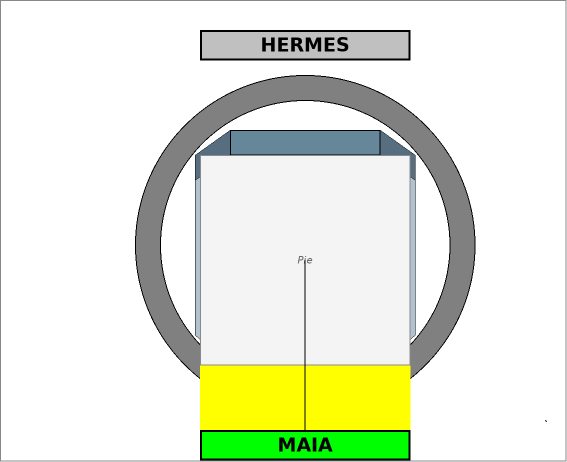
VISUALIZATION VISU_M3RotationFigure_1  // 567x462
    Ellipse (135,75 340x340)
    Ellipse (160,100 290x290)
    Polygon (545,420) (546,421)
    Polygon (230,155) (195,180) (195,155) (230,130) (380,130) (415,155) (415,180) (380,155)
    Polygon (230,365) (195,335) (195,180) (230,155) (380,155) (415,180) (415,335) (380,365)
    Line (565,390)
    Rectangle (230,130 150x25)
    Rectangle (200,260 210x200)
    Pie (200,155 210x210)
    Line (305,445) (305,260)
    Rectangle (200,430 210x30), "MAIA"
    Rectangle (200,30 210x30), "HERMES"
END_VISUALIZATION

(* stored: Version 1.1.0.1, ProductVersion 3.1.4019.2
   Visu VISU_M3RotationFigure_1: Id {22ddfc68-cfd6-4f28-9f31-a8ac68a89a1e} *)
